FUNCTION FUN_SCALE : REAL
VAR_INPUT
	ix : REAL;
	ixmax : REAL;
	ixmin : REAL;
	rymax : REAL;
	rymin : REAL;
END_VAR
VAR
	rk : REAL := 0;
	rd : REAL := 0;
END_VAR

rk := (rymax - rymin)/(ixmax - ixmin);
rd := rymin - rk * ixmin;

FUN_SCALE := rk * ix + rd;

IF FUN_SCALE > rymax THEN
	FUN_SCALE := rymax;
ELSIF FUN_SCALE < rymin THEN
	FUN_SCALE := rymin;
END_IF

END_FUNCTION

(* stored: Version 1.1.0.1, ProductVersion 3.1.4024.15
   POU FUN_SCALE: Id {504b1975-0664-4c3b-a385-d2e4730a72fe}, SpecialFunc None *)
